PROGRAM FlowCheck
VAR_INPUT
	start : BOOL := FALSE;
	setSpeedDuration : TIME := T#15S;
	runTestDuration : TIME := T#15S;
	runTestWeight : lreal := 10.0; // run for 100 grams
	autoAdvance : BOOL := TRUE;
END_VAR
VAR_OUTPUT
	startTimes : ARRAY[1..50] OF ULINT;
	endTimes : ARRAY[1..50] OF ULINT;
	FQA : ARRAY[1..50] OF LREAL;
	FQB : ARRAY[1..50] OF LREAL;
	FQC : ARRAY[1..50] OF LREAL;
	weight : ARRAY[1..50] OF LREAL;
	FTA_mean : ARRAY[1..50] OF LREAL;
	FTB_mean : ARRAY[1..50] OF LREAL;
	FTC_mean : ARRAY[1..50] OF LREAL;
	P9999Atubing : ARRAY[1..50] OF INT;
	P9999Btubing : ARRAY[1..50] OF INT;
END_VAR
VAR
	i : UINT := 0; // index
	n : UINT := 25;
	t : LREAL := 0.0;
	tol : LREAL := 5.0;
	//spA : ARRAY [1..50] OF LREAL := [10.0, 20.0, 30.0, 40.0, 50.0, 60.0, 70.0, 80.0, 90.0, 100.0, 
    //                                125.0, 150.0, 175.0, 200.0, 225.0, 250.0, 275.0, 300.0,
    //                                350.0, 400.0, 450.0, 500.0, 550.0, 600.0,
	//								0.0,0.0,0.0,0.0,0.0,0.0,0.0,0.0,0.0,0.0,0.0,0.0,0.0,0.0,0.0,0.0,0.0,0.0,0.0,0.0,0.0,0.0,0.0,0.0];
	spA : ARRAY [1..50] OF LREAL := [10.0, 20.0, 30.0, 40.0, 50.0, 60.0, 70.0, 80.0, 90.0, 100.0, 
                                    110.0, 120.0, 130.0, 140.0, 150.0, 0.0, 0.0, 0.0,
                                    0.0, 0.0, 0.0, 0.0, 0.0, 0.0,
									0.0,0.0,0.0,0.0,0.0,0.0,0.0,0.0,0.0,0.0,0.0,0.0,0.0,0.0,0.0,0.0,0.0,0.0,0.0,0.0,0.0,0.0,0.0,0.0];
	spB : ARRAY [1..50] OF LREAL := [0.0,0.0,0.0,0.0,0.0,0.0,0.0,0.0,0.0,0.0,0.0,0.0,0.0,0.0,0.0,0.0,0.0,0.0,0.0,0.0,0.0,0.0,0.0,0.0,
									0.0,0.0,0.0,0.0,0.0,0.0,0.0,0.0,0.0,0.0,0.0,0.0,0.0,0.0,0.0,0.0,0.0,0.0,0.0,0.0,0.0,0.0,0.0,0.0
	];
	//								0.0, 20.0, 30.0, 40.0, 50.0, 60.0, 70.0, 80.0, 90.0, 100.0, 
    //                                125.0, 150.0, 175.0, 200.0, 225.0, 250.0, 275.0, 300.0,
    //                                350.0, 400.0, 450.0, 500.0, 550.0, 600.0];
	//spA : ARRAY [1..50] OF LREAL := [0.0,0.0,0.0,0.0,0.0,0.0,0.0,0.0,0.0,0.0,0.0,0.0,0.0,0.0,0.0,0.0,0.0,0.0,0.0,0.0,0.0,0.0,0.0,0.0,
	//								0.0, 20.0, 30.0, 40.0, 50.0, 60.0, 70.0, 80.0, 90.0, 100.0, 
    //                                125.0, 150.0, 175.0, 200.0, 225.0, 250.0, 275.0, 300.0,
    //                                350.0, 400.0, 450.0, 500.0, 550.0, 600.0];
	//sp : ARRAY [1..50] OF LREAL := [51.0, 58.0, 64.0, 79.0, 97.0, 112.0, 128.0, 151.0, 210.0, 280.0, 335.0, 410.0, 480.0, 600.0];
	//sp : ARRAY [1..50] OF LREAL := [335.0, 410.0, 480.0, 600.0];
	setSpeed : SFCStepType;
	runTest : SFCStepType;
	recordTest : SFCStepType;
END_VAR

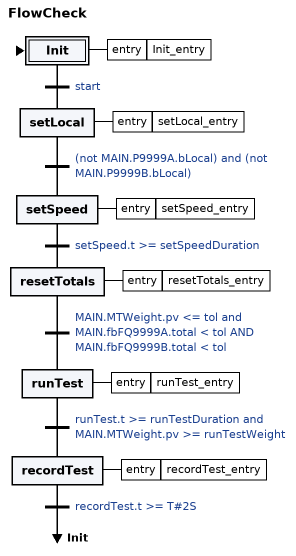
INITIAL_STEP Init:
    Init_entry(P1);  // entry action
END_STEP
TRANSITION FROM Init TO setLocal
    := start;
END_TRANSITION
STEP setLocal:
    setLocal_entry(P1);  // entry action
END_STEP
TRANSITION FROM setLocal TO setSpeed
    := (not MAIN.P9999A.bLocal) and (not MAIN.P9999B.bLocal);
END_TRANSITION
STEP setSpeed:
    setSpeed_entry(P1);  // entry action
END_STEP
TRANSITION FROM setSpeed TO resetTotals
    := setSpeed.t >= setSpeedDuration;
END_TRANSITION
STEP resetTotals:
    resetTotals_entry(P1);  // entry action
END_STEP
TRANSITION FROM resetTotals TO runTest
    := MAIN.MTWeight.pv <= tol and MAIN.fbFQ9999A.total < tol AND MAIN.fbFQ9999B.total < tol;
END_TRANSITION
STEP runTest:
    runTest_entry(P1);  // entry action
END_STEP
TRANSITION FROM runTest TO recordTest
    := runTest.t >= runTestDuration and MAIN.MTWeight.pv >= runTestWeight;
END_TRANSITION
STEP recordTest:
    recordTest_entry(P1);  // entry action
END_STEP
TRANSITION FROM recordTest TO Init
    := recordTest.t >= T#2S;
END_TRANSITION

ACTION Init_entry:
IF i >= n THEN
	MAIN.P9999A.nRun_RQ := 0; //stop pump
	MAIN.P9999B.nRun_RQ := 0; //stop pump
	start := FALSE;
	i := 0;
END_IF
MAIN.logActive := FALSE;
END_ACTION

ACTION resetTotals_entry:
MAIN.fbFQ9999A.resetRQ := TRUE;
MAIN.fbFQ9999B.resetRQ := TRUE;
MAIN.fbFQ9999C.resetRQ := TRUE;
MAIN.MTSendString := 'ZI$0D$0A';
MAIN.logActive := TRUE;
END_ACTION

ACTION setSpeed_entry:
i := i + 1;
startTimes[i] := 0;
endTimes[i] := 0;
FQA[i] := 0;
FQB[i] := 0;
FQC[i] := 0;
weight[i] := 0;
FTA_mean[i] := 0;
FTB_mean[i] := 0;
FTC_mean[i] := 0;
IF spA[i] > 0.1 THEN
	MAIN.P9999A.nRun_RQ := 1; //start pump
	MAIN.P9999A.fSpeedSP_RQ := spA[i];
ELSE
	MAIN.P9999A.nRun_RQ := 0; //stop pump
	MAIN.P9999A.fSpeedSP_RQ := 0.0;
END_IF
	
IF spB[i] > 0.1 THEN
	MAIN.P9999B.nRun_RQ := 1; //start pump
	MAIN.P9999B.fSpeedSP_RQ := spB[i];
ELSE
	MAIN.P9999B.nRun_RQ := 0; //stop pump
	MAIN.P9999B.fSpeedSP_RQ := 0.0;
END_IF

P9999Atubing[i] := MAIN.P9999A.nTubeSize;
P9999Btubing[i] := MAIN.P9999B.nTubeSize;
END_ACTION

ACTION setLocal_entry:
IF MAIN.P9999A.bLocal THEN
	MAIN.P9999A.nLocal_RQ := 0;  //put pump in remote
END_IF
IF MAIN.P9999B.bLocal THEN
	MAIN.P9999B.nLocal_RQ := 0;  //put pump in remote
END_IF
END_ACTION

ACTION recordTest_entry:
endTimes[i] := unixTime;
FQA[i] := MAIN.fbFQ9999A.total;
FQB[i] := MAIN.fbFQ9999B.total;
FQC[i] := MAIN.fbFQ9999C.total;
weight[i] := MAIN.MTWeight.pv;
t := DWORD_TO_LREAL(TIME_TO_DWORD(runTestDuration))/1000.0/60.0;
FTA_mean[i] := MAIN.fbFQ9999A.total/t;
FTB_mean[i] := MAIN.fbFQ9999B.total/t;
FTC_mean[i] := MAIN.fbFQ9999C.total/t;
IF NOT autoAdvance THEN
	start := FALSE;
END_IF
END_ACTION

ACTION runTest_entry:
MAIN.MTSendString := 'SIR$0D$0A';
startTimes[i] := unixTime;
END_ACTION

END_PROGRAM

(* stored: Version 1.1.0.1, ProductVersion 3.1.0.36
   POU FlowCheck: Id {5af3dc8a-7e5a-4711-bca5-17d71c2a26ea}, SpecialFunc None
   Action Init_entry: Id {2c7f0757-376b-4664-8340-64e21c1687ac}
   Action resetTotals_entry: Id {42e03fb6-3cc9-4d62-bfe7-006a7768173a}
   Action setSpeed_entry: Id {848cd76c-d321-45a4-b4a4-715fef5a0e03}
   Action setLocal_entry: Id {b55c3b40-24b5-4d93-acf5-8ede72550ec4}
   Action recordTest_entry: Id {bde3d7fd-3957-4ac5-8388-8d931f021eff}
   Action runTest_entry: Id {c81ced17-7403-423d-b9f6-ed0097e4666c} *)
